FUNCTION_BLOCK FB_RobotRegionMove_BufferArea EXTENDS FB_ObjectBase_V2 IMPLEMENTS IBasicElement
VAR_INPUT
    Robot : REFERENCE TO FB_FanucRobot_Basic;
    // Command   : ST_WareHouseWithRobotMove_Command;
    Info : ST_RobotRegionMove_Info;
    Stop : BOOL;
END_VAR
VAR_OUTPUT
    // Status : ST_WareHouseWithRobotMove_Status;

END_VAR
VAR
    _Abort       : BOOL;
    strStatus    : STRING;
    uiResumeStep : UINT;

    Area : E_RobotArea := E_RobotArea.BufferArea;
    UseA : BOOL;
    UseB : BOOL;

    Get               : BOOL;
    tonTimeOut        : TON;
    _UniqueErrorCode  : STRING;
    PreviousStrStatus : STRING;
    PreviousErrorCode : STRING;
END_VAR

SUPER^.A10_StateControl();
A00_BasicUnits();

METHOD M_CheckCommand : BOOL // True : Command is useful
VAR_INPUT
END_VAR
VAR
	
END_VAR
// Check command paremeter is correct

THIS^.Get :=Info.Get;
UseA := Info.UseA;
UseB := Info.UseB;
//Buffer area
		
		IF UseA AND ( Info.A_Position<1 OR  Info.A_Position>40) THEN
			strStatus:='Wrong command ,Position A Not allow';
			M_CheckCommand:=FALSE;
			RETURN;			
		END_IF		
	
		IF UseB AND( Info.B_Position<1 OR  Info.B_Position>40 )THEN
			strStatus:='Wrong command ,Position B Not allow';
			M_CheckCommand:=FALSE;
			RETURN;			
		END_IF
		
M_CheckCommand:=TRUE;
END_METHOD

METHOD M_CheckUnitsNotBusy : BOOL
VAR_INPUT
END_VAR
M_CheckUnitsNotBusy := true;
END_METHOD

METHOD M_CheckUnitsReady : BOOL
VAR_INPUT
END_VAR
M_CheckUnitsReady := true;
END_METHOD

METHOD  M_STATE_ABORTED
VAR_INPUT
END_VAR
ERROR :=TRUE;
Busy    := FALSE;
Aborted := TRUE;
Status := strStatus;
UniqueErrorCode:=_UniqueErrorCode;
IF NOT Execute THEN
	eSTATE:=STATE_RESETTING;
END_IF

IF Execute AND Reset THEN
	uiExecutingStep :=uiResumeStep;
	PreviousStrStatus := strStatus;
	PreviousErrorCode := _UniqueErrorCode;
	eSTATE:=STATE_EXECUTING;
END_IF
END_METHOD

METHOD  M_STATE_ABORTING
VAR_INPUT
END_VAR
CASE uiAbortingStep OF
	0 :
		uiAbortingStep:=9999;
		IF strStatus = PreviousStrStatus THEN
			_UniqueErrorCode :=PreviousErrorCode;
		END_IF
		_Abort :=FALSE;
	9999:	_AbortCompleted:=TRUE;
END_CASE

IF _AbortCompleted THEN	
	eSTATE :=STATE_ABORTED;
END_IF
END_METHOD

METHOD  M_STATE_DONE
VAR_INPUT
END_VAR
Busy := FALSE;
Done := TRUE;
IF NOT Execute THEN
    eState := STATE_RESETTING;
END_IF
END_METHOD

METHOD  M_STATE_DORMANT
VAR_INPUT
END_VAR
// Clear FB output
Busy            := FALSE;
Done            := FALSE;
Aborted         := FALSE;
Error           := FALSE;
ErrorID         := 0;
Status          := '';
_ResetCompleted := FALSE;
_Error          := FALSE;
_Executed       := FALSE;

tonTimeOut.IN:=FALSE;
strStatus :='No Error';
uiExecutingStep :=uiResettingStep :=uiResumeStep :=0;
PreviousStrStatus			 :='';
PreviousErrorCode			 :='';
_UniqueErrorCode	:='0';

// Wait Execute command
IF Execute THEN
    eState := STATE_EXECUTING;
END_IF
END_METHOD

METHOD  M_STATE_ERROR
VAR_INPUT
END_VAR
ERROR   :=TRUE;
Busy	:=FALSE;
Status := strStatus;
UniqueErrorCode:=_UniqueErrorCode;
IF NOT Execute THEN	
eSTATE:=STATE_RESETTING;
END_IF
END_METHOD

METHOD  M_STATE_EXECUTING
VAR_INPUT
END_VAR
VAR_INST
    ActionMode       : E_ReloadRoundBoxAction;
	BoxReady_1st : BOOL;
	BoxReady_2nd : BOOL;
    CarrierReady_1st : BOOL;
    CarrierReady_2nd : BOOL;
    uiBothStep : UINT;
    uiSingleClampStep : UINT;
	Address_A : INT;
	Address_B : INT;
END_VAR
VAR
	WareHouse: INT;
END_VAR
// Set Busy active edit by johnson
Busy := TRUE;
IF THIS^.Stop THEN // Pending the timeout when Stop signal occur
	tonTimeout.IN :=FALSE;
END_IF
// Service Process
CASE uiExecutingStep OF
	0:
        // Clear variable
        ActionMode       := E_ReloadRoundBoxAction.Undefined;
        CarrierReady_1st := FALSE;
        CarrierReady_2nd := FALSE;
        uiBothStep := 0;
		uiSingleClampStep :=0;
		BoxReady_1st := 0;
		BoxReady_2nd := 0;
		tonTimeOut.IN:=FALSE;
        // Check command
        IF M_CheckCommand() THEN
            uiExecutingStep := 10;
		ELSE
			_Error:=TRUE;
        END_IF
    10:
        // Start process, check units first
        IF M_CheckUnitsReady() THEN
            uiExecutingStep := 20;
        END_IF
    20:
        // CHeck units not busy state
        IF M_CheckUnitsNotBusy() THEN
            uiExecutingStep := 1000;
        END_IF
   
	1000:   
			// Read   coordinate
 			 Address_A := LREAL_TO_INT(Info.A_Position);
			 Address_B := LREAL_TO_INT(Info.B_Position);
			 
			IF UseA AND NOT UseB THEN
				//Only clampA
				uiExecutingStep := 10000;
			ELSIF NOT UseA AND UseB THEN
				//Only ClampB 
				uiExecutingStep := 20000;
			ELSIF UseA AND UseB THEN
				//Both Clamps
				uiExecutingStep := 30000;		
			END_IF
       
    10000: // Only ClampA 
        IF NOT Robot._DI1.Done THEN            
           		BoxReady_1st:=TRUE;				
			          		 
				  // Robot Abs move
           		 Robot.M_StartRobotAbsMove(GetBox:=Get,
											UseClampA:=UseA,
											UseClampB:=UseB,
											Area:=Area,
											ClampA_Address:=Address_A,
											ClampB_Address:=Address_B,
											BoxReady_1:=BoxReady_1st,
											BoxReady_2:=BoxReady_2nd);	  
		
        ELSE
			tonTimeOut.IN:=FALSE;
            uiExecutingStep := 10080;
        END_IF
			tonTimeOut.IN:=TRUE;
			IF tonTimeOut.Q=TRUE THEN
				tonTimeOut.IN:=FALSE;			
				strStatus :='Reset Robot timeout';
				_Error:=TRUE;
			END_IF	
    10080:
        Robot.M_ResetRobotAbsMove(UseA,UseB); // Clear command and go to place box
		tonTimeOut.IN:=TRUE;
        IF NOT Robot._DI1.Done THEN
			tonTimeOut.IN:=FALSE;
            uiExecutingStep := 99000; 
        END_IF
    	IF tonTimeOut.Q=TRUE THEN
			strStatus :='Reset Robot timeout';
			_Error:=TRUE;
		END_IF	
    
   20000: // Only ClampB
        IF NOT Robot._DI1.Done THEN           		
				BoxReady_2nd:=TRUE;				          		 
				  // Robot Abs move
           		 Robot.M_StartRobotAbsMove( GetBox:=Get,
											UseClampA:=UseA,
											UseClampB:=UseB,
											Area:=Area,
											ClampA_Address:=Address_A,
											ClampB_Address:=Address_B,
											BoxReady_1:=BoxReady_1st,
											BoxReady_2:=BoxReady_2nd);	
        ELSE
			tonTimeOut.IN:=FALSE;
            uiExecutingStep := 20080;
        END_IF
		tonTimeOut.IN:=TRUE;
			IF tonTimeOut.Q=TRUE THEN
				tonTimeOut.IN:=FALSE;			
				strStatus :='Reset Robot timeout';
				_Error:=TRUE;
			END_IF	
    20080:
       Robot.M_ResetRobotAbsMove(UseA,UseB);; // Clear command 

        IF NOT Robot._DI1.Done THEN
            uiExecutingStep := 99000; 
        END_IF
		tonTimeOut.IN:=TRUE;
		IF tonTimeOut.Q=TRUE THEN
			strStatus :='Reset Robot timeout';
			_Error:=TRUE;
		END_IF	
    30000: // Both Clamps
        		
		
		  CASE uiBothStep OF
           		0://	
					BoxReady_1st := FALSE;
					BoxReady_2nd := FALSE;					
					uiBothStep:=1000;	
	
				1000:
						BoxReady_1st:=TRUE;
						uiBothStep:=2000;
						
				2000:
						IF Robot._DI1.Notification THEN
							uiBothStep:=3000;
						END_IF
				3000:
					
					
						uiBothStep:=9000;	
					
				9000:
						BoxReady_2nd:=TRUE;
						uiBothStep:=9999;
				
				9999: //Wait		
        // wait reset
        END_CASE

       	  // Robot Abs move
           		 Robot.M_StartRobotAbsMove( GetBox:=Get,
											UseClampA:=UseA,
											UseClampB:=UseB,
											Area:=Area,
											ClampA_Address:=Address_A,
											ClampB_Address:=Address_B,
											BoxReady_1:=BoxReady_1st,
											BoxReady_2:=BoxReady_2nd);	
		
		
        IF Robot._DI1.Done THEN
			tonTimeOut.IN:=FALSE;
            uiExecutingStep := 30080;
        END_IF
		IF tonTimeOut.Q=TRUE THEN
				tonTimeOut.IN:=FALSE;			
				strStatus :='Reset Robot timeout';
				_Error:=TRUE;
			END_IF	
    30080: // Check robot command is clear
        
        Robot.M_ResetRobotAbsMove(UseA,UseB);

        IF NOT Robot._DI1.Done THEN
			tonTimeOut.IN:=FALSE;
            uiExecutingStep := 99000; // go to place step
        END_IF    
   		tonTimeOut.IN:=TRUE;
		IF tonTimeOut.Q=TRUE THEN
			strStatus :='Stop Robot timeout';
			_Error:=TRUE;
		END_IF	
   
    99000: // process done
                Status    := 'Process completed';
        _Executed := TRUE;
END_CASE

IF _Executed THEN
    eState := STATE_DONE;
ELSIF _Error THEN
	//FUN_UniqueErrorCodeGenerator(iErrorID := ErrorID,UinqueErrorCode=>_UniqueErrorCode);
    eState := STATE_ERROR;
ELSIF NOT Execute THEN
    eState := STATE_RESETTING;
END_IF
IF _Abort OR Abort THEN
	//FUN_UniqueErrorCodeGenerator(iErrorID := ErrorID,UinqueErrorCode=>_UniqueErrorCode);
	eSTATE:=STATE_ABORTING;
END_IF
END_METHOD

METHOD  M_STATE_RESETTING
VAR_INPUT
END_VAR
Error :=FALSE;
Done :=FALSE;
Busy := FALSE;


CASE uiResettingStep OF
	
	0:
		tonTimeOut.IN:=FALSE;
		Robot.M_ResetAllCommand();
		Robot.M_ResetRobotAbsMove(TRUE,TRUE);
		
		uiResettingStep:=9999;
	9999:
		_ResetCompleted:=TRUE;
END_CASE
IF _ResetCompleted THEN
	eSTATE:=STATE_DORMANT;
END_IF
END_METHOD

END_FUNCTION_BLOCK

(* stored: Version 1.1.0.1, ProductVersion 3.1.4024.13
   POU FB_RobotRegionMove_BufferArea: Id {6cc52740-03ba-469a-b8b4-856268bb0152}, SpecialFunc None
   Folder Method: Id {8c8868d7-0097-4403-9c44-eebf62295eba}
   Folder State: Id {d387bd16-6c2f-4235-8036-17b925fb6f8b}
   Method M_CheckCommand: Id {fa8748bd-e370-4888-a902-cb916f4ae882}
   Method M_CheckUnitsNotBusy: Id {20ac2ea1-2b04-4f7a-b4eb-c8068b0ef2cf}
   Method M_CheckUnitsReady: Id {f153be14-3203-4a5f-aa37-f7b6915b9c33}
   Method M_STATE_ABORTED: Id {9c1a8684-ec55-4de0-a1e6-6f4781c45742}
   Method M_STATE_ABORTING: Id {364ba5c4-8b28-455a-a26d-4f6aa4ea3d12}
   Method M_STATE_DONE: Id {a8edbefe-d075-4e38-9f9b-d2c0937154b2}
   Method M_STATE_DORMANT: Id {4444f06f-f50d-4703-94d1-bfdecfbfeb52}
   Method M_STATE_ERROR: Id {577204b3-103d-4210-aab3-69f65a1363ee}
   Method M_STATE_EXECUTING: Id {027645c3-4b49-4dc2-992b-dc3c95343a88}
   Method M_STATE_RESETTING: Id {ef94a4f5-0f6c-45eb-84cf-7c468bfbc761} *)
